Staubli VAL3: refreshStatic.pgx

program refreshStatic()
  local string l_sMessage[2]
  local string l_sMenu
  local string l_sSession
begin
  cls()
  //
  gotoxy(1,1)
  put("F2  AXIS7")
  gotoxy(1,3)
  put("F4  AXIS8")
  gotoxy(5,13)
  put("AXIS7")
  gotoxy(15,13)
  put("AXIS8")
  //
end
